PROGRAM MAIN
VAR
	_station001 : Station001;
END_VAR

_station001.Run();

END_PROGRAM

(* stored: Version 1.1.0.1, ProductVersion 3.1.4024.6
   POU MAIN: Id {e5777d28-b709-40e2-b696-3956f2b85f68}, SpecialFunc None *)
